// TIA Portal V20 export
FUNCTION_BLOCK "Simulation"   // FB196, LAD
// stored: MemoryReserve 100, Namespace Unit1.Em12, SetENOAutomatically false
   VAR_INPUT
      simulation { ExternalAccessible := 'False'; ExternalVisible := 'False'; ExternalWritable := 'False'} : Bool;
   END_VAR
   VAR
      instActuator { ExternalAccessible := 'False'; ExternalVisible := 'False'; ExternalWritable := 'False'} : Array[0..9] of "Simulation_Actuator";
   END_VAR
BEGIN

REGION Network 1: Actuator
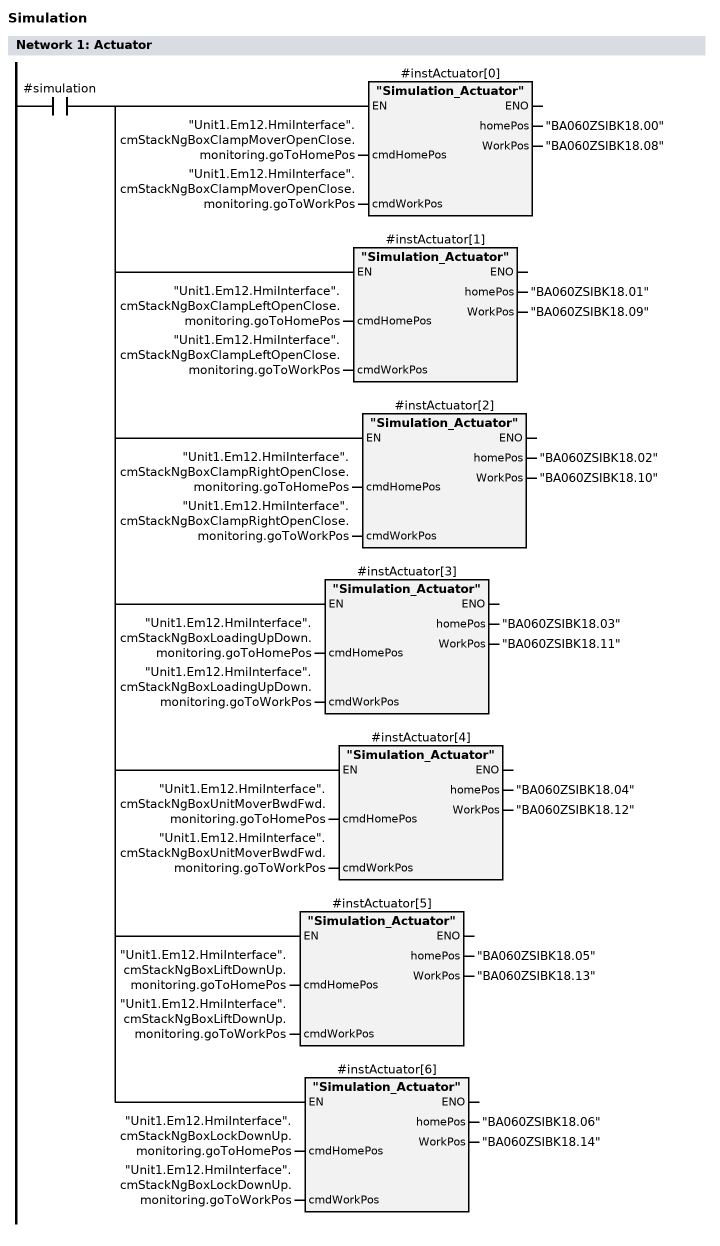
   RUNG wire#powerrail
      Contact( #simulation )
      wire#w1
      #instActuator[0](cmdHomePos := "Unit1.Em12.HmiInterface".cmStackNgBoxClampMoverOpenClose.monitoring.goToHomePos, cmdWorkPos := "Unit1.Em12.HmiInterface".cmStackNgBoxClampMoverOpenClose.monitoring.goToWorkPos, homePos => "BA060ZSIBK18.00", WorkPos => "BA060ZSIBK18.08")
   END_RUNG
   RUNG wire#w1
      #instActuator[1](cmdHomePos := "Unit1.Em12.HmiInterface".cmStackNgBoxClampLeftOpenClose.monitoring.goToHomePos, cmdWorkPos := "Unit1.Em12.HmiInterface".cmStackNgBoxClampLeftOpenClose.monitoring.goToWorkPos, homePos => "BA060ZSIBK18.01", WorkPos => "BA060ZSIBK18.09")
   END_RUNG
   RUNG wire#w1
      #instActuator[2](cmdHomePos := "Unit1.Em12.HmiInterface".cmStackNgBoxClampRightOpenClose.monitoring.goToHomePos, cmdWorkPos := "Unit1.Em12.HmiInterface".cmStackNgBoxClampRightOpenClose.monitoring.goToWorkPos, homePos => "BA060ZSIBK18.02", WorkPos => "BA060ZSIBK18.10")
   END_RUNG
   RUNG wire#w1
      #instActuator[3](cmdHomePos := "Unit1.Em12.HmiInterface".cmStackNgBoxLoadingUpDown.monitoring.goToHomePos, cmdWorkPos := "Unit1.Em12.HmiInterface".cmStackNgBoxLoadingUpDown.monitoring.goToWorkPos, homePos => "BA060ZSIBK18.03", WorkPos => "BA060ZSIBK18.11")
   END_RUNG
   RUNG wire#w1
      #instActuator[4](cmdHomePos := "Unit1.Em12.HmiInterface".cmStackNgBoxUnitMoverBwdFwd.monitoring.goToHomePos, cmdWorkPos := "Unit1.Em12.HmiInterface".cmStackNgBoxUnitMoverBwdFwd.monitoring.goToWorkPos, homePos => "BA060ZSIBK18.04", WorkPos => "BA060ZSIBK18.12")
   END_RUNG
   RUNG wire#w1
      #instActuator[5](cmdHomePos := "Unit1.Em12.HmiInterface".cmStackNgBoxLiftDownUp.monitoring.goToHomePos, cmdWorkPos := "Unit1.Em12.HmiInterface".cmStackNgBoxLiftDownUp.monitoring.goToWorkPos, homePos => "BA060ZSIBK18.05", WorkPos => "BA060ZSIBK18.13")
   END_RUNG
   RUNG wire#w1
      #instActuator[6](cmdHomePos := "Unit1.Em12.HmiInterface".cmStackNgBoxLockDownUp.monitoring.goToHomePos, cmdWorkPos := "Unit1.Em12.HmiInterface".cmStackNgBoxLockDownUp.monitoring.goToWorkPos, homePos => "BA060ZSIBK18.06", WorkPos => "BA060ZSIBK18.14")
   END_RUNG
   // the same network as SCL:
   IF #simulation THEN
       #instActuator[0](cmdHomePos := "Unit1.Em12.HmiInterface".cmStackNgBoxClampMoverOpenClose.monitoring.goToHomePos,   // "Simulation_Actuator"
                        cmdWorkPos := "Unit1.Em12.HmiInterface".cmStackNgBoxClampMoverOpenClose.monitoring.goToWorkPos,
                        homePos => "BA060ZSIBK18.00",
                        WorkPos => "BA060ZSIBK18.08");
       #instActuator[1](cmdHomePos := "Unit1.Em12.HmiInterface".cmStackNgBoxClampLeftOpenClose.monitoring.goToHomePos,   // "Simulation_Actuator"
                        cmdWorkPos := "Unit1.Em12.HmiInterface".cmStackNgBoxClampLeftOpenClose.monitoring.goToWorkPos,
                        homePos => "BA060ZSIBK18.01",
                        WorkPos => "BA060ZSIBK18.09");
       #instActuator[2](cmdHomePos := "Unit1.Em12.HmiInterface".cmStackNgBoxClampRightOpenClose.monitoring.goToHomePos,   // "Simulation_Actuator"
                        cmdWorkPos := "Unit1.Em12.HmiInterface".cmStackNgBoxClampRightOpenClose.monitoring.goToWorkPos,
                        homePos => "BA060ZSIBK18.02",
                        WorkPos => "BA060ZSIBK18.10");
       #instActuator[3](cmdHomePos := "Unit1.Em12.HmiInterface".cmStackNgBoxLoadingUpDown.monitoring.goToHomePos,   // "Simulation_Actuator"
                        cmdWorkPos := "Unit1.Em12.HmiInterface".cmStackNgBoxLoadingUpDown.monitoring.goToWorkPos,
                        homePos => "BA060ZSIBK18.03",
                        WorkPos => "BA060ZSIBK18.11");
       #instActuator[4](cmdHomePos := "Unit1.Em12.HmiInterface".cmStackNgBoxUnitMoverBwdFwd.monitoring.goToHomePos,   // "Simulation_Actuator"
                        cmdWorkPos := "Unit1.Em12.HmiInterface".cmStackNgBoxUnitMoverBwdFwd.monitoring.goToWorkPos,
                        homePos => "BA060ZSIBK18.04",
                        WorkPos => "BA060ZSIBK18.12");
       #instActuator[5](cmdHomePos := "Unit1.Em12.HmiInterface".cmStackNgBoxLiftDownUp.monitoring.goToHomePos,   // "Simulation_Actuator"
                        cmdWorkPos := "Unit1.Em12.HmiInterface".cmStackNgBoxLiftDownUp.monitoring.goToWorkPos,
                        homePos => "BA060ZSIBK18.05",
                        WorkPos => "BA060ZSIBK18.13");
       #instActuator[6](cmdHomePos := "Unit1.Em12.HmiInterface".cmStackNgBoxLockDownUp.monitoring.goToHomePos,   // "Simulation_Actuator"
                        cmdWorkPos := "Unit1.Em12.HmiInterface".cmStackNgBoxLockDownUp.monitoring.goToWorkPos,
                        homePos => "BA060ZSIBK18.06",
                        WorkPos => "BA060ZSIBK18.14");
   END_IF;
END_REGION

REGION Network 2 (SCL)
   IF #simulation AND "JB_Temp".Test_Homing[12] THEN

       "Unit1.Em12.HmiInterface".cmStackNgBoxLoadingUpDown.commands.commandHomePos :=
       "Unit1.Em12.HmiInterface".cmStackNgBoxClampLeftOpenClose.commands.commandHomePos :=
       "Unit1.Em12.HmiInterface".cmStackNgBoxClampRightOpenClose.commands.commandHomePos :=
       "Unit1.Em12.HmiInterface".cmStackNgBoxLiftDownUp.commands.commandHomePos :=
       "Unit1.Em12.HmiInterface".cmStackNgBoxLockDownUp.commands.commandWorkPos := true;
       "Unit1.Em12.HmiInterface".cmStackNgBoxUnitMoverBwdFwd.commands.commandWorkPos := true;

       "JB_Temp".Test_Homing[12] := false;

   END_IF;

   IF #simulation AND "JB_Temp".Test_Homing[20] THEN

       "Unit1.Em12.HmiInterface".cmStackNgBoxLoadingUpDown.commands.commandHomePos :=
       "Unit1.Em12.HmiInterface".cmStackNgBoxClampLeftOpenClose.commands.commandHomePos :=
       "Unit1.Em12.HmiInterface".cmStackNgBoxClampRightOpenClose.commands.commandHomePos :=
       "Unit1.Em12.HmiInterface".cmStackNgBoxLiftDownUp.commands.commandHomePos :=
       "Unit1.Em12.HmiInterface".cmStackNgBoxLockDownUp.commands.commandWorkPos := FALSE;
       "Unit1.Em12.HmiInterface".cmStackNgBoxUnitMoverBwdFwd.commands.commandWorkPos := FALSE;

   END_IF;
END_REGION
END_FUNCTION_BLOCK
